// TwinCAT 3 PLC project main
// ProgramVersion: 3.1.4024.0
// libraries:
//   Tc2_BABasic, * (Beckhoff Automation GmbH)
//   Tc2_Standard, * (Beckhoff Automation GmbH)
//   Tc2_System, * (Beckhoff Automation GmbH)
//   Tc3_Module, * (Beckhoff Automation GmbH)
// project tree:
//   / GlobalTextList.TcGTLO, PlcTask.TcTTO, Visualization Manager.TcVMO (not stored)
//   POUs/ MAIN.TcPOU
//   VISUs/ Visu.TcVIS
// real-time tasks:
//   TASK PlcTask: cycle T#10ms, priority 20, ADS port 350

CONFIGURATION main
    RESOURCE PLC ON TwinCAT3
        TASK PlcTask(INTERVAL := T#10ms, PRIORITY := 20);
        PROGRAM MAIN WITH PlcTask : MAIN;
    END_RESOURCE
END_CONFIGURATION

// ---- POUs/MAIN.TcPOU
PROGRAM MAIN
VAR
	//Variabelen
	bAllesAan : BOOL;
	bAllesUit : BOOL;
	
	//Druktoetsen
	bDrukVoorduer : BOOL;
	bDrukKeuken1 : BOOL;
	bDrukKeuekn2 : BOOL;
	bDrukLiving1a : BOOL;
	bDrukLiving1b : BOOL;
	bDrukLiving2a : BOOL;
	bDrukLiving2b : BOOL;
	
	//Lichten
	bLichtKeueken : BOOL;
	bLichtLiving1 : BOOL;
	bLichtLiving2 : BOOL;
	
	//Functie blokken
	fbLichtKeueken : FB_Light;
	fbLichtLiving1 : FB_Light;
	fbLichtLiving2 : FB_Light;
	
	fbLankKlikAlleUit : FB_ShortLongClick;
	fbDubbelKlikAlleAan : FB_SingleDoubleClick;
END_VAR

fbDubbelKlikAlleAan(
	bSwitch := bDrukVoorduer,
	tSwitchTime := T#2S,
	bDoubleClick => bAllesUit
);

fbLankKlikAlleUit(
	bSwitch := bDrukVoorduer,
	tSwitchTime := T#5S,
	bLongClick => bAllesUit
);

fbLichtKeueken(
	bOn := bAllesAan,
	bOff := bAllesUit,
	bToggle := bDrukKeuken1 OR bDrukKeuekn2,
	bLight => bLichtKeueken
);

fbLichtLiving1(
	bOn := bAllesAan,
	bOff := bAllesUit,
	bToggle := bDrukLiving1a OR bDrukLiving2b,
	bLight => bLichtLiving1
);

fbLichtLiving2(
	bOn := bAllesAan,
	bOff := bAllesUit,
	bToggle := bDrukLiving1b OR bDrukLiving2a,
	bLight => bLichtLiving2
);

END_PROGRAM

// ---- GlobalTextList.TcGTLO
TEXTLIST GlobalTextList
  220 = 'bDrukKeuken1'
  804 = 'bDrukKeuken2'
  367 = 'bDrukLiving1a'
  582 = 'bDrukLiving1b'
  964 = 'bDrukLiving2a'
  648 = 'bDrukLiving2b'
  605 = 'bDrukVoordeur'
  204 = 'bLichtKeuken'
  986 = 'bLichtLiving1'
  47 = 'bLichtLiving2'
  533 = 'Label'
END_TEXTLIST

// ---- VISUs/Visu.TcVIS
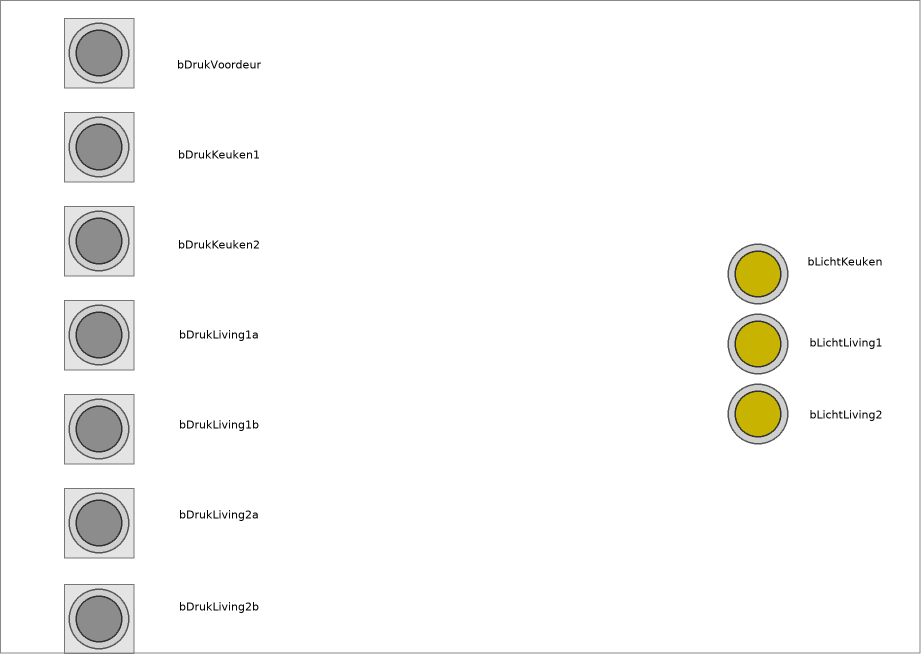
VISUALIZATION Visu  // 921x654
    PushSwitch (64,18 70x70), variable: MAIN.bDrukVoorduer, behaviour: TAP, style: Switch-PushSwitch-Gray
    PushSwitch (64,584 70x70), variable: MAIN.bDrukLiving2b, behaviour: TAP, style: Switch-PushSwitch-Gray
    PushSwitch (64,488 70x70), variable: MAIN.bDrukLiving2a, behaviour: TAP, style: Switch-PushSwitch-Gray
    PushSwitch (64,112 70x70), variable: MAIN.bDrukKeuken1, behaviour: TAP, style: Switch-PushSwitch-Gray
    PushSwitch (64,206 70x70), variable: MAIN.bDrukKeuekn2, behaviour: TAP, style: Switch-PushSwitch-Gray
    PushSwitch (64,300 70x70), variable: MAIN.bDrukLiving1a, behaviour: TAP, style: Switch-PushSwitch-Gray
    PushSwitch (64,394 70x70), variable: MAIN.bDrukLiving1b, behaviour: TAP, style: Switch-PushSwitch-Gray
    Lamp1 (723,239 70x70), variable: MAIN.bLichtKeueken, style: Lamp-Lamp1-Yellow
    Lamp1 (723,309 70x70), variable: MAIN.bLichtLiving1, style: Lamp-Lamp1-Yellow
    Lamp1 (723,379 70x70), variable: MAIN.bLichtLiving2, style: Lamp-Lamp1-Yellow
    Label (144,320 150x30), "bDrukLiving1a"
    Label (770,247 150x30), "bLichtKeuken"
    Label (144,140 150x30), "bDrukKeuken1"
    Label (144,230 150x30), "bDrukKeuken2"
    Label (144,592 150x30), "bDrukLiving2b"
    Label (144,410 150x30), "bDrukLiving1b"
    Label (144,500 150x30), "bDrukLiving2a"
    Label (144,50 150x30), "bDrukVoordeur"
    Label (771,328 150x30), "bLichtLiving1"
    Label (771,400 150x30), "bLichtLiving2"
END_VISUALIZATION
